FUNCTION_BLOCK FINAL SpindleDeltaVFDOverEIP IMPLEMENTS SpindleController
VAR
	// Delta VFD control for the spindle
	oSpindleControl AT %Q* : ST_DeltaVFDCommandWord;
	oSpindleFrequency AT %Q* : UINT;
END_VAR
VAR CONSTANT
	// Number of RPM per HZ in the VFD
	RPMPerHZ : UINT := 30;
	// VFD frequency precision in 1/X of 1 HZ. So 10 means it can do 1/10th of a HZ
	VFDHZPrecision : UINT := 10;
	// Minimum VFD RPM increment based on RPM per HZ and precision
	VFDMinRPMIncrement : UINT := TO_UINT(RPMPerHZ / VFDHZPrecision);
END_VAR

METHOD Run : BOOL
oSpindleControl.Stop := FALSE;
oSpindleControl.Run := TRUE;
END_METHOD

METHOD SetDirection : BOOL
VAR_INPUT
	// Set the spindle rotation direction
	Reverse	: BOOL;
END_VAR
IF Reverse THEN
	oSpindleControl.Reverse := TRUE;
	oSpindleControl.Forward := FALSE;
ELSE
	oSpindleControl.Reverse := FALSE;
	oSpindleControl.Forward := TRUE;
END_IF
END_METHOD

METHOD SetSpeed : BOOL
VAR_INPUT
	Speed: UINT;
END_VAR
// The spindle frequency is in increments of 0.1hz
oSpindleFrequency := (SPEED * Constants.VFDHZPrecision) / Constants.RPMPerHZ;
END_METHOD

METHOD Stop : BOOL
oSpindleControl.Stop := TRUE;
oSpindleControl.Run := FALSE;
END_METHOD

END_FUNCTION_BLOCK

(* stored: Version 1.1.0.1, ProductVersion 3.1.4022.16
   POU SpindleDeltaVFDOverEIP: Id {6020789a-138f-4f2b-90da-86ac6f55afbb}, SpecialFunc None
   Method Run: Id {f7dbc088-ec96-4dc7-82a4-4e3a10cc37b0}
   Method SetDirection: Id {1359955e-6c76-49de-b255-f132b5eba728}
   Method SetSpeed: Id {551c4af6-92c1-4681-a2be-40253c4c3b04}
   Method Stop: Id {089f55cd-61cf-48b3-8afe-f2aa50859904} *)
